// TIA Portal V20 export
TYPE "typeHmiParameter"
// stored: Access Published, Namespace Unit1
   STRUCT
      General { S7_SetPoint := 'True'} : "Unit1.typeHmiParameterParameters";
      EM0 { S7_SetPoint := 'True'} : "Unit1.typeHmiParameterParameters";
      EM1 { S7_SetPoint := 'True'} : "Unit1.typeHmiParameterParameters";
      EM2 { S7_SetPoint := 'True'} : "Unit1.typeHmiParameterParameters";
      EM3 { S7_SetPoint := 'True'} : "Unit1.typeHmiParameterParameters";
      EM4 { S7_SetPoint := 'True'} : "Unit1.typeHmiParameterParameters";
      EM5 { S7_SetPoint := 'True'} : "Unit1.typeHmiParameterParameters";
      EM6 { S7_SetPoint := 'True'} : "Unit1.typeHmiParameterParameters";
      EM7 { S7_SetPoint := 'True'} : "Unit1.typeHmiParameterParameters";
      FFU_Parameter { S7_SetPoint := 'True'} : Array[1..18] of "HMI_IF_Parameter_Parameter_UDT";
      Save_BT { S7_SetPoint := 'True'} : "HMI_IF_Parameter_Save Button_UDT";
   END_STRUCT;
   // // General.Data[0] : CPM
   // // General.Data[1] : Anode Electrode Width
   // // General.Data[2] : Cathode Electrode Width
   // // General.Data[3] : Anode Tab Width
   // // General.Data[4] : Cathode Tab Width
   // // General.Data[5] : Anode Electrode ~ TabWidth
   // // General.Data[6] : Cathode Electrode ~ TabWidth
   // // General.Data[7] : Anode Gap Width
   // // General.Data[8] : Cathode Gap Width
   // // General.Data[9] : Anode Thinkness
   // // General.Data[10] : Cathode Thinkness
   // // General.Data[11] : Separator Thinkness
   // // General.Data[12] : Jelly Roll Width
   // // General.Data[13] : Cell Stack Count
   // // EM3.Data[21] : TargetDancerAngle
   // // EM3.Data[22] : DancerLenth
   // // EM3.Data[23] : Compasator Storke
END_TYPE
